// SIMATIC S7-200 project (STEP 7-Micro/WIN), CPU 224 REL 01.11

ORGANIZATION_BLOCK MAIN:OB1
TITLE=主PLC通过PPI协议向远程PLC发送控制指令。
// 系统在首次上电时，设置为PPI主站模式，并清空相关数据区。
// 运行过程中，系统在每个1秒脉冲的上升沿，整理发送数据缓冲区，设置远程站地址、数据地址指针和数据长度，递增发送数据，并通过NETW指令发送至远程PLC。
// 在1秒脉冲的下降沿，且特定条件满足时，系统设置远程站地址、数据地址指针和数据长度，通过NETR指令从远程PLC读取数据至接收数据缓冲区。
// 之后，在常开标志为1时，PLC将接收数据移动至输出字，用于显示远程反应釜的状态。
BEGIN
Network 1 // 网络标题
// 开机时定义本机为ppi主站（否则缺省为从站）
// 清空v区数据
LD     SM0.1
MOVB   2, SMB30
FILL   +0, VW100, 100
?000
Network 2 // 数据发送
// 在每个1s脉冲的上升沿，整理数据表头，并发送数据。
// 远程的站地址为6；
// 对方接收数据的开始地址为vb0；
// 共发送2个byte；
// 生成数据vw107递增，对应远程的vb0；
// 发送命令执行。
// 
LD     SM0.5
EU
MOVB   6, VB101
MOVD   &VB0, VD102
MOVB   2, VB106
INCW   VW107
?233   VB100, 0
Network 3 // 数据接收
// 在1s脉冲的下降沿接收数据；
// 远程站地址6；
// 从远程vb0开始读取；
// 长度8个字节；
// 读取命令执行
LD     SM0.5
ED
AN     SM0.1
AN     V100.6
AN     V100.5
MOVB   6, VB201
MOVD   &VB0, VD202
MOVB   8, VB206
?232   VB200, 0
Network 4 // 收到的数据显示
// 其实对应远程的vw4
// 207,208,209,210,211.......
// 0,1,2,3,4.......
LD     SM0.0
MOVW   VW211, QW0
END_ORGANIZATION_BLOCK
